TYPE EL3403_PM_Outputs :
STRUCT
	{attribute addProperty Name "Index"}
	Index AT %Q* : USINT;
END_STRUCT
END_TYPE

(* stored: Version 1.1.0.1, ProductVersion 3.1.4024.9
   DUT EL3403_PM_Outputs: Id {2fabaa5e-b57e-0ac2-395a-feb589cd8bd2} *)
